FUNCTION_BLOCK T_RoboConnect_SetAnalogOutput_CorrectIndexPasses EXTENDS T_UnitTestBase
VAR
  robot : I_RoboConnect;
  targetDO : UINT;
  myTestState, prevState :
    (INIT, ARRANGE, ACT, ASSERT) := INIT;
  expected, actual : BOOL;
  counter : UINT;
END_VAR

CASE myTestState OF
  INIT:
    StateChanged();
    myTestState := ARRANGE;

  ARRANGE:
    IF StateChanged() THEN
      expected := TRUE;
      myTestSTate := ACT;
    END_IF

  ACT:
    actual := robot.SetAnalogOutput(targetDO, 0.5);
    myTestState := ASSERT;

  ASSERT:
    assertion.AssertEquals_BOOL(expected, actual, 'robot.SetAnalogOutput(targetDO,TRUE)');
    TestFinished();
    myTestState := INIT;

END_CASE

METHOD FB_init : BOOL
VAR_INPUT
  bInitRetains : BOOL; // if TRUE, the retain variables are initialized (warm start / cold start)
  bInCopyCode : BOOL; // if TRUE, the instance afterwards gets moved into the copy code (online change)
  TestSuite : tcl_SimpleUnitTestLibrary.I_TestSuite;
  robot : I_TcRobot;
  targetDo : UINT;
END_VAR
THIS^.robot := robot;
THIS^.targetDo := targetDo;
END_METHOD

METHOD PRIVATE StateChanged : BOOL
IF  myTestState = prevState THEN
  RETURN;
END_IF

prevState := myTestState;
StateChanged := TRUE;
END_METHOD

METHOD WaitForCycles : BOOL
VAR_INPUT
  maxCount : UINT;
END_VAR
counter := counter + 1;

IF counter = maxCount THEN
  counter := 0;
  WaitForCycles := TRUE;
END_IF
END_METHOD

END_FUNCTION_BLOCK

(* stored: Version 1.1.0.1
   POU T_TcRobot_SetAnalogOutput_CorrectIndexPasses: Id {42e06875-d387-435b-8009-989327393191}, SpecialFunc None
   Method FB_init: Id {fc6f34cf-0875-4f7f-b43c-5ab6d3c11d02}
   Method StateChanged: Id {d43f4fec-46bc-4e4c-8195-0a848e7b47bf}
   Method WaitForCycles: Id {13a867ca-b4d7-4c26-b872-84bd041f5cfb} *)
